PROGRAM TestRunner
VAR
END_VAR

END_PROGRAM

(* stored: Version 1.1.0.1
   POU TestRunner: Id {67416dad-cafd-42c9-a195-e92f9a1c42b6}, SpecialFunc None *)
